// SIMATIC STEP 7 (V5.x) project PompesSysteme
// CPU: CPU313 C-2 DP(1)
// station: P_ADR_BUS
// station: Hardware
// station: SIMATIC 300 Station
// program: S7 Program(1)

SYMBOL_TABLE
"MonFB1"	FB 1	FB 1	// Description de MonFB1
"G7_STD_3"	FC 72	FC 72
"b1"	I 0.1	BOOL	// Position basse 1
"b2"	I 0.2	BOOL	// Position basse 2
"b3"	I 0.3	BOOL	// Position basse 3
"h1"	I 0.4	BOOL	// Position haute 1
"h2"	I 0.5	BOOL	// Position haute 2
"h3"	I 0.6	BOOL	// Position haute 3
"Cycle Execution"	OB 1	OB 1	// Programme principale
"Complete Restart"	OB 100	OB 100	// Initiation des variables
"P1"	Q 0.1	BOOL	// Marche pompe 1
"P2"	Q 0.2	BOOL	// Marche pompe 2
"P3"	Q 0.3	BOOL	// Marche pompe 3
"TIME_TCK"	SFC 64	SFC 64	// Read the System Time
END_SYMBOL_TABLE

FUNCTION_BLOCK "MonFB1"	// FB 1
TITLE = S7GRAPH V4 FB
//Block fonctionnel des pompes - GRAFCET
VERSION : 0.1
VAR_INPUT
  OFF_SQ : BOOL ;
  INIT_SQ : BOOL ;
  ACK_EF : BOOL ;
  S_PREV : BOOL ;
  S_NEXT : BOOL ;
  SW_AUTO : BOOL ;
  SW_TAP : BOOL ;
  SW_MAN : BOOL ;
  S_SEL : INT ;
  S_ON : BOOL ;
  S_OFF : BOOL ;
  T_PUSH : BOOL ;
END_VAR
VAR_OUTPUT
  S_NO : INT ;
  S_MORE : BOOL ;
  S_ACTIVE : BOOL ;
  ERR_FLT : BOOL ;
  AUTO_ON : BOOL ;
  TAP_ON : BOOL ;
  MAN_ON : BOOL ;
END_VAR
VAR
  G7T : ARRAY  [0 .. 6 ] OF STRUCT
   TV : BOOL ;
   TT : BOOL ;
   TS : BOOL ;
   CF_IV : BOOL ;
   TNO : INT ;
   CRIT : DWORD ;
   CRIT_OLD : DWORD ;
   CRIT_FLT : DWORD ;
  END_STRUCT ;
  G7S : ARRAY  [0 .. 4 ] OF STRUCT
   S1 : BOOL ;
   L1 : BOOL ;
   V1 : BOOL ;
   R1 : BOOL ;
   A1 : BOOL ;
   S0 : BOOL ;
   L0 : BOOL ;
   V0 : BOOL ;
   X : BOOL ;
   LA : BOOL ;
   VA : BOOL ;
   RA : BOOL ;
   AA : BOOL ;
   SS : BOOL ;
   LS : BOOL ;
   VS : BOOL ;
   SNO : INT ;
   T : TIME ;
   U : TIME ;
   CRIT_LOC : DWORD ;
   CRIT_LOC_ERR : DWORD ;
   CRIT_SUP : DWORD ;
   SM : BOOL ;
   LP : BOOL ;
   LN : BOOL ;
   VP : BOOL ;
   VN : BOOL ;
   H_IL_ERR : BYTE ;
   H_SV_FLT : BYTE ;
   RESERVED : DWORD ;
  END_STRUCT ;
  TVX : ARRAY  [0 .. 6 ] OF BYTE  := B#16#1;
  TTX : ARRAY  [0 .. 6 ] OF BYTE  := B#16#1;
  TSX : ARRAY  [0 .. 2 ] OF BYTE  := B#16#1;
  S00X : ARRAY  [0 .. 2 ] OF BYTE  := B#16#1;
  SOFFX : ARRAY  [0 .. 2 ] OF BYTE  := B#16#1;
  SONX : ARRAY  [0 .. 2 ] OF BYTE  := B#16#1;
  SAX : ARRAY  [0 .. 2 ] OF BYTE  := B#16#1;
  SERRX : ARRAY  [0 .. 5 ] OF BYTE  := B#16#1;
  SMX : ARRAY  [0 .. 5 ] OF BYTE  := B#16#1;
  S0X : ARRAY  [0 .. 5 ] OF BYTE  := B#16#1;
  S1X : ARRAY  [0 .. 5 ] OF BYTE  := B#16#1;
  S_DISPLAY : INT ;
  S_SEL_OLD : INT ;
  S_DISPIDX : BYTE ;
  T_DISPIDX : BYTE ;
  MOPEDGE : STRUCT
   AUTO : BOOL ;
   MAN : BOOL ;
   TAP : BOOL ;
   TOP : BOOL ;
   RES1 : BOOL ;
   RES2 : BOOL ;
   RES3 : BOOL ;
   RES4 : BOOL ;
   LOCK : BOOL ;
   SUP : BOOL ;
   ACKREQ : BOOL ;
   SSKIP : BOOL ;
   OFF : BOOL ;
   INIT : BOOL ;
   HALT : BOOL ;
   TMS_HALT : BOOL ;
   OPS_ZERO : BOOL ;
   SACT_DISP : BOOL ;
   SEF_DISP : BOOL ;
   SALL_DISP : BOOL ;
   S_PREV : BOOL ;
   S_NEXT : BOOL ;
   S_SELOK : BOOL ;
   S_ON : BOOL ;
   S_OFF : BOOL ;
   T_PUSH : BOOL ;
   REG : BOOL ;
   ACK : BOOL ;
   IL_PERM : BOOL ;
   T_PERM : BOOL ;
   ILP_MAN : BOOL ;
  END_STRUCT ;
  MOP : STRUCT
   AUTO : BOOL  := TRUE;
   MAN : BOOL ;
   TAP : BOOL ;
   TOP : BOOL ;
   RES1 : BOOL ;
   RES2 : BOOL ;
   RES3 : BOOL ;
   RES4 : BOOL ;
   LOCK : BOOL  := TRUE;
   SUP : BOOL  := TRUE;
   ACKREQ : BOOL  := TRUE;
   SSKIP : BOOL ;
   OFF : BOOL ;
   INIT : BOOL  := TRUE;
   HALT : BOOL ;
   TMS_HALT : BOOL ;
   OPS_ZERO : BOOL ;
   SACT_DISP : BOOL  := TRUE;
   SEF_DISP : BOOL ;
   SALL_DISP : BOOL ;
   S_PREV : BOOL ;
   S_NEXT : BOOL ;
   S_SELOK : BOOL ;
   S_ON : BOOL ;
   S_OFF : BOOL ;
   T_PUSH : BOOL ;
   REG : BOOL ;
   ACK : BOOL ;
   IL_PERM : BOOL ;
   T_PERM : BOOL ;
   ILP_MAN : BOOL ;
  END_STRUCT ;
  TICKS : STRUCT
   DELTA : TIME ;
   OLD : TIME ;
   NEW : TIME ;
  END_STRUCT ;
  SQ_FLAGS : STRUCT
   ERR_FLT : BOOL ;
   ERROR : BOOL ;
   FAULT : BOOL ;
   RT_FAIL : BOOL ;
   NO_SNO : BOOL ;
   NF_OFL : BOOL ;
   SA_OFL : BOOL ;
   TV_OFL : BOOL ;
   MSG_OFL : BOOL ;
   NO_SWI : BOOL ;
   CYC_OP : BOOL ;
   AS_MSG : BOOL ;
   AS_SEND : BOOL ;
   SQ_BUSY : BOOL ;
   SA_BUSY : BOOL ;
   AS_SIG : BOOL ;
  END_STRUCT ;
  S_PTR : DWORD  := DW#16#3D0;
  S_PTR2 : DWORD ;
  S_PTR3 : DWORD  := DW#16#A80;
  S_PTR4 : DWORD  := DW#16#A50;
  T_PTR : DWORD  := DW#16#A20;
  C_AR2 : DWORD ;
  M_FBDB : DWORD  := DW#16#10000;
  M_SNO : WORD ;
  M_EVID : WORD ;
  M_EVIL : DWORD ;
  M_EVSV : DWORD ;
  M_EV : DWORD  := DW#16#990;
  CRIT : ARRAY  [0 .. 31 ] OF BOOL ;
  S_START : BYTE ;
  S_IDX : BYTE ;
  S_INT : INT  := 72;
  S_TMP : BYTE ;
  T_START : BYTE ;
  T_IDX : BYTE ;
  T_TMP : BYTE ;
  T_TMP2 : BYTE ;
  TV_POT : BYTE  := B#16#6;
  RETURN1 : BYTE ;
  RETURN2 : BYTE ;
  SINI : ARRAY  [0 .. 2 ] OF BYTE  := B#16#2, B#16#1;
  LSTT : ARRAY  [0 .. 6 ] OF BYTE  := B#16#0, B#16#0, B#16#0, B#16#0, B#16#3, B#16#1, B#16#2;
  ATAJ : ARRAY  [0 .. 6 ] OF BYTE  := B#16#0, B#16#1, B#16#2, B#16#3, B#16#4, B#16#5, B#16#6;
  ATAB : ARRAY  [0 .. 6 ] OF BYTE  := B#16#0, B#16#1, B#16#5, B#16#6, B#16#4, B#16#2, B#16#3;
  PSTT : ARRAY  [0 .. 6 ] OF BYTE  := B#16#0, B#16#1, B#16#2, B#16#3, B#16#4, B#16#2, B#16#3;
  NSTT : ARRAY  [0 .. 6 ] OF BYTE  := B#16#1, B#16#2, B#16#3, B#16#4, B#16#3, B#16#1, B#16#2;
  ASSJ : ARRAY  [0 .. 4 ] OF BYTE  := B#16#0, B#16#1, B#16#2, B#16#3, B#16#4;
  ASSB : ARRAY  [0 .. 4 ] OF BYTE  := B#16#0, B#16#1, B#16#2, B#16#3, B#16#4;
  PTTS : ARRAY  [0 .. 4 ] OF BYTE  := B#16#0, B#16#0, B#16#1, B#16#2, B#16#3;
  NTTS : ARRAY  [0 .. 4 ] OF BYTE  := B#16#0, B#16#1, B#16#2, B#16#3, B#16#4;
  PRE_CNT : WORD ;
  POST_CNT : WORD ;
  ADR_COND : WORD ;
  MAX_TVAL : BYTE  := B#16#5;
  MAX_SACT : BYTE  := B#16#1;
  MAX_CRIT : BYTE  := B#16#4;
  T_CNT : BYTE  := B#16#6;
  SUP_CNT : BYTE ;
  LOCK_CNT : BYTE ;
  S_CNT : BYTE  := B#16#4;
  SQ_CNT : BYTE  := B#16#1;
  PRS_INPAR : DWORD  := DW#16#E000F6C8;
  PRS_OUTPAR : DWORD  := DW#16#E000800D;
  GC_FLAGS : STRUCT
   T_MACH : WORD  := W#16#EB;
   COND_ED : WORD  := W#16#E3;
   W_LEVEL : WORD  := W#16#D5;
   AS_MSG : WORD ;
   FB_IF : WORD  := W#16#FC;
   SSB : WORD  := W#16#105;
   CRIT_AVAIL : BOOL ;
   SSKIP_AVAIL : BOOL  := TRUE;
   SSKIP_ON : BOOL ;
   ACK_REQ : BOOL  := TRUE;
   SYNC_AVAIL : BOOL ;
   ILP_MAN : BOOL ;
  END_STRUCT ;
  G7_FBMARK : BYTE  := B#16#25;
  G7_RELEASE : BYTE  := B#16#2A;
  G7_ID2 : BYTE  := B#16#37;
  G7_ID1 : BYTE  := B#16#47;
END_VAR
BEGIN
// body was compiled from an S7-GRAPH chart; compiled code not shown
END_FUNCTION_BLOCK

// FC 72: know-how protected block, not included

DATA_BLOCK DB 1
VERSION : 0.0
"MonFB1"
BEGIN
END_DATA_BLOCK

ORGANIZATION_BLOCK "Cycle Execution"	// OB 1
TITLE = "Main Program Sweep (Cycle)"
VERSION : 0.1
VAR_TEMP
  OB1_EV_CLASS : BYTE ;	//Bits 0-3 = 1 (Coming event), Bits 4-7 = 1 (Event class 1)
  OB1_SCAN_1 : BYTE ;	//1 (Cold restart scan 1 of OB 1), 3 (Scan 2-n of OB 1)
  OB1_PRIORITY : BYTE ;	//Priority of OB Execution
  OB1_OB_NUMBR : BYTE ;	//1 (Organization block 1, OB1)
  OB1_RESERVED_1 : BYTE ;	//Reserved for system
  OB1_RESERVED_2 : BYTE ;	//Reserved for system
  OB1_PREV_CYCLE : INT ;	//Cycle time of previous OB1 scan (milliseconds)
  OB1_MIN_CYCLE : INT ;	//Minimum cycle time of OB1 (milliseconds)
  OB1_MAX_CYCLE : INT ;	//Maximum cycle time of OB1 (milliseconds)
  OB1_DATE_TIME : DATE_AND_TIME ;	//Date and time OB1 started
END_VAR
BEGIN
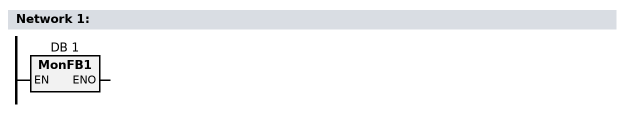
NETWORK
TITLE =
      CALL  "MonFB1" , DB 1;
      NOP   0;
END_ORGANIZATION_BLOCK

ORGANIZATION_BLOCK "Complete Restart"	// OB 100
TITLE = "Complete Restart"
VERSION : 0.1
VAR_TEMP
  OB100_EV_CLASS : BYTE ;	//16#13, Event class 1, Entering event state, Event logged in diagnostic buffer
  OB100_STRTUP : BYTE ;	//16#81/82/83/84 Method of startup
  OB100_PRIORITY : BYTE ;	//Priority of OB Execution
  OB100_OB_NUMBR : BYTE ;	//100 (Organization block 100, OB100)
  OB100_RESERVED_1 : BYTE ;	//Reserved for system
  OB100_RESERVED_2 : BYTE ;	//Reserved for system
  OB100_STOP : WORD ;	//Event that caused CPU to stop (16#4xxx)
  OB100_STRT_INFO : DWORD ;	//Information on how system started
  OB100_DATE_TIME : DATE_AND_TIME ;	//Date and time OB100 started
END_VAR
BEGIN
// (block stored without names or comments; labels and parameter names are numbered)
END_ORGANIZATION_BLOCK
